ABB RobotStudio station: Práctica2.rsstn

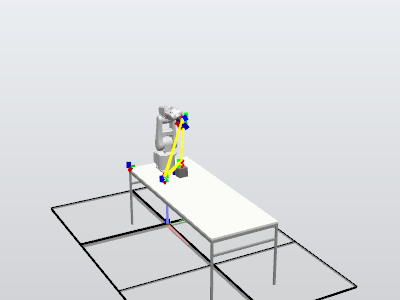
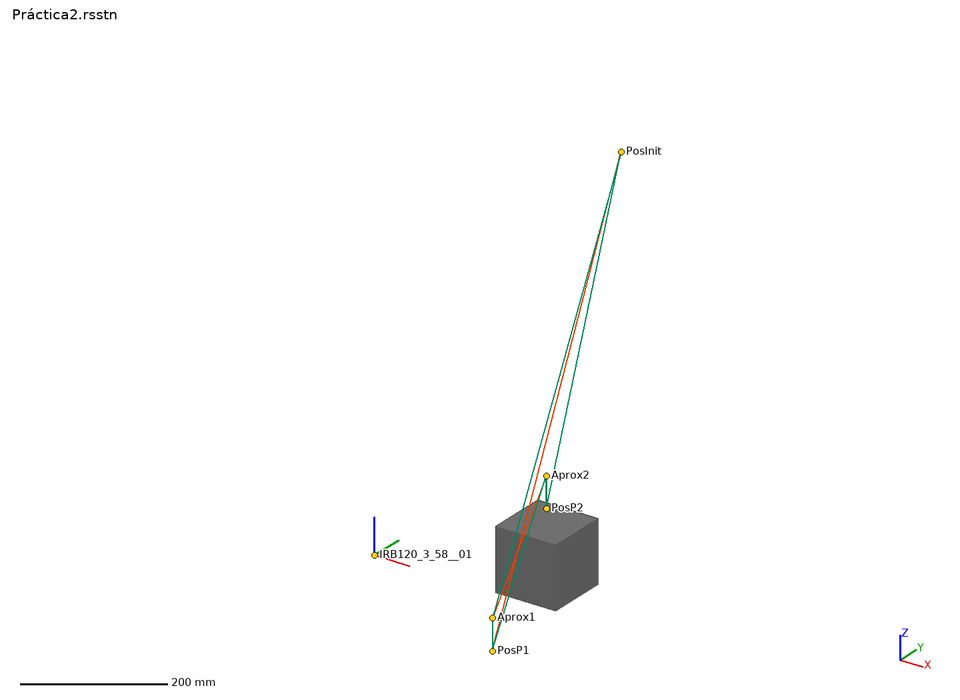
[picture v1: parts stored in the station drawn from their meshes, with robot base, taught points and paths (robot models come from the ABB library and are not in the file)]
Station Práctica2 (saved by RobotStudio 25.1.11133.0)
Controller Controlador2, task T_ROB1: task frame (RAPID world) sits at (0, 0, 670) mm in the station
Controller Controlador2
  mechanical unit ROB_1: IRB120_3_58__01, 6 joints, base frame (0, 0, 0) mm
Layout (positions relative to the parent item):
  - TVentosa [mechanism] at (341.72, -4.33, 1323.66) mm, rotated rx -155.61 ry 54.34 rz -134.33 deg
      TCP TVentosa at (0, 0, 51.19) mm
      links: Mi_herramienta
  - LogicGate [smart component, from Components\LogicGate.rslib]
      properties: Operator=NOT; Delay=0
  - LogicGate_2 [smart component, from Components\LogicGate.rslib]
      properties: Operator=AND; Delay=0
  - IRB120_3_58__01 [mechanism, from %ABB.RobotStudio.Models.IRB120%\IRB120_3_58_G_01.rslib] at (0, 0, 670) mm; joint values [-0.0763, 0.013, -0.2247, 0.415, 0.8466, -0.7718] (rad or m)
  - table [part, from Downloads\Table.rslib] at (-200, 350, 669.71) mm, rotated rx 0 ry 0 rz -90 deg
  - Pieza_1 [part], size 50 x 30 x 20 mm
  - Pieza_2 [part] at (200, 0, 670) mm, size 100 x 100 x 100 mm
  - CollisionSensor_2 [smart component, from Components\CollisionSensor.rslib]
      properties: Object1=TVentosa; Object2=Pieza_1; NearMiss=0.001; Part1=(none); Part2=(none); CollisionType=0
  - Attacher_2 [smart component, from Components\Attacher.rslib]
      properties: Parent=Detacher_2; Flange=0; Child=Pieza_1; Mount=true; Offset=[0 0 0]; Orientation=[0 0 0]
  - Detacher_2 [smart component, from Components\Detacher.rslib]
      properties: Child=Pieza_1; KeepPosition=true
Attachment: TVentosa is attached to IRB120_3_58__01 / Link6
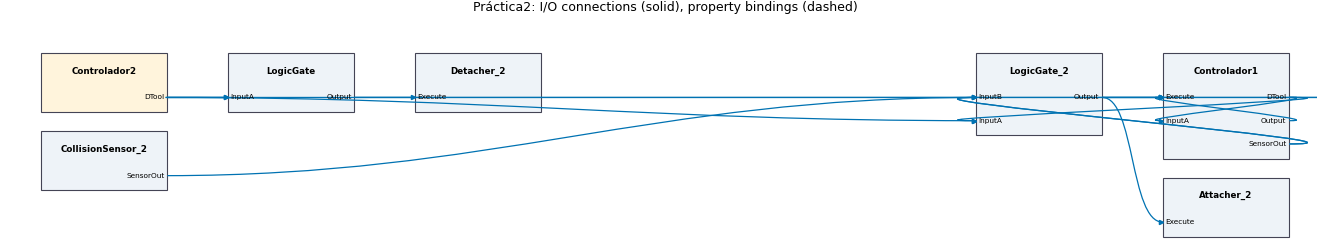
Station logic (signal -> signal, property => property):
  Controlador1.DTool -> Attacher.Execute
  Controlador1.DTool -> LogicGate_2.InputA
  LogicGate_2.Output -> Detacher.Execute
  Controlador1.DTool -> LogicGate.InputA
  LogicGate.Output -> Detacher.Execute
  CollisionSensor.SensorOut -> LogicGate_2.InputB
  Controlador1.DTool -> LogicGate_2.InputA
  LogicGate_2.Output -> Attacher.Execute
  Controlador2.DTool -> LogicGate_2.InputA
  CollisionSensor.SensorOut -> LogicGate_2.InputB
  LogicGate_2.Output -> Attacher.Execute
  CollisionSensor_2.SensorOut -> LogicGate_2.InputB
  LogicGate_2.Output -> Attacher_2.Execute
  Controlador2.DTool -> LogicGate.InputA
  LogicGate.Output -> Detacher_2.Execute
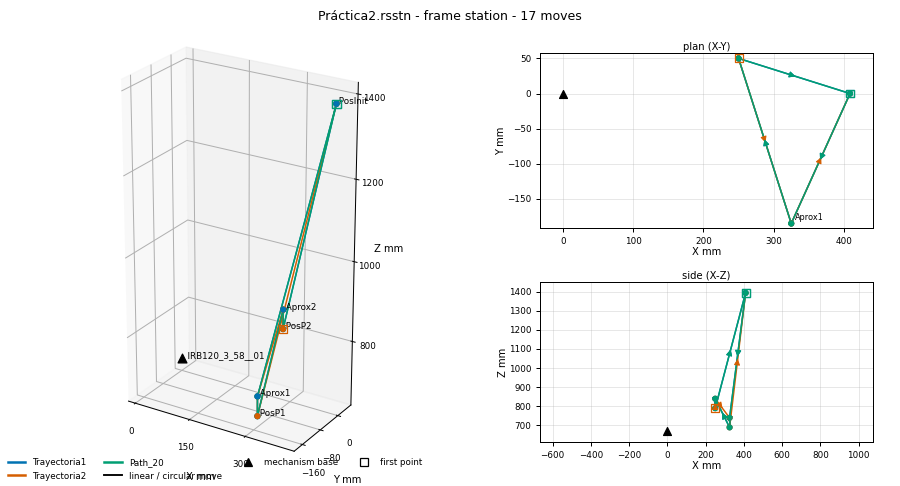
[picture p0: tool path of Práctica2.rsstn in frame station, 17 of 17 moves have a stored position in this frame; points joined in program order, loops and branches not executed]
Targets, tools, work objects and paths stored in the station, written as RAPID:
! task T_ROB1
MODULE CalibData
  PERS tooldata TVentosa:=[TRUE,[[0,0,51.19],[1,0,0,0]],[0.1,[0,0,1],[1,0,0,0],0,0,0]];
  TASK PERS wobjdata WO_Pieza1:=[FALSE,TRUE,"",[[-200,-350,-0.292],[1,0,0,0]],[[500,150,0.292],[1,0,0,0]]];
  TASK PERS wobjdata WO_Pieza2:=[FALSE,TRUE,"",[[-200,-350,-0.292],[1,0,0,0]],[[400,350,0.292],[1,0,0,0]]];
ENDMODULE

! task T_ROB1
MODULE Module1
  CONST robtarget Aprox1:=[[25,15,70],[0,0,1,0],[-1,0,-1,0],[9E+09,9E+09,9E+09,9E+09,9E+09,9E+09]];
  CONST robtarget PosP1:=[[25,15,20],[0,0,1,0],[-1,0,-1,0],[9E+09,9E+09,9E+09,9E+09,9E+09,9E+09]];
  CONST robtarget PosP2:=[[50,50,120],[0,1,0,0],[0,0,-2,0],[9E+09,9E+09,9E+09,9E+09,9E+09,9E+09]];
  CONST robtarget Aprox2:=[[50,50,170],[0,1,0,0],[0,0,-2,0],[9E+09,9E+09,9E+09,9E+09,9E+09,9E+09]];
  CONST robtarget PosInit:=[[408.686,0,722.885],[0.5,0,0.866025404,0],[0,0,0,0],[9E+09,9E+09,9E+09,9E+09,9E+09,9E+09]];
  CONST robtarget Target_70:=[[408.686,0,722.885],[0.500000007,0,0.8660254,0],[0,0,0,0],[9E+09,9E+09,9E+09,9E+09,9E+09,9E+09]];
  CONST robtarget Target_20:=[[25,15,70],[0,0,1,0],[-1,0,-1,0],[9E+09,9E+09,9E+09,9E+09,9E+09,9E+09]];
  CONST robtarget Target_30:=[[25,15,20],[0,0,1,0],[-1,0,-1,0],[9E+09,9E+09,9E+09,9E+09,9E+09,9E+09]];
  CONST robtarget Target_50:=[[50,50,170],[0,1,0,0],[0,0,-2,0],[9E+09,9E+09,9E+09,9E+09,9E+09,9E+09]];
  CONST robtarget Target_40:=[[50,50,120],[0,1,0,0],[0,0,-2,0],[9E+09,9E+09,9E+09,9E+09,9E+09,9E+09]];
  PROC Trayectoria1()
    MoveL PosInit,v500,z100,TVentosa\WObj:=wobj0;
    MoveL Aprox1,v500,z100,TVentosa\WObj:=WO_Pieza1;
    MoveL PosP1,v500,fine,TVentosa\WObj:=WO_Pieza1;
    SetDO DTool,1;
    WaitTime 0.5;
    MoveL Aprox2,v500,z100,TVentosa\WObj:=WO_Pieza2;
    MoveL PosP2,v500,fine,TVentosa\WObj:=WO_Pieza2;
    SetDO DTool,0;
    WaitTime 0.5;
    MoveL PosInit,v500,z100,TVentosa\WObj:=wobj0;
  ENDPROC
  PROC Trayectoria2()
    MoveL PosP2,v500,fine,TVentosa\WObj:=WO_Pieza2;
    MoveL Aprox2,v500,z100,TVentosa\WObj:=WO_Pieza2;
    MoveL Aprox1,v500,z100,TVentosa\WObj:=WO_Pieza1;
    MoveL PosP1,v500,fine,TVentosa\WObj:=WO_Pieza1;
    MoveL PosInit,v500,z100,TVentosa\WObj:=wobj0;
  ENDPROC
  PROC main()
    Trayectoria1;
    Trayectoria2;
  ENDPROC
  PROC Path_20()
    MoveL Target_70,v500,z100,TVentosa\WObj:=wobj0;
    MoveL Target_20,v500,z100,TVentosa\WObj:=WO_Pieza1;
    MoveL Target_30,v500,fine,TVentosa\WObj:=WO_Pieza1;
    MoveL Target_50,v500,z100,TVentosa\WObj:=WO_Pieza2;
    MoveL Target_40,v500,fine,TVentosa\WObj:=WO_Pieza2;
    MoveL Target_70,v500,z100,TVentosa\WObj:=wobj0;
  ENDPROC
ENDMODULE

